// Brief: setup Arm Joint3-5 decelerate to stop
FUNCTION_BLOCK PUBLIC FB_SetupCtrlStop EXTENDS FB_SetupArmCtrlBase
VAR
	// stop motion is terminated after set time period
	m_maxStopPeriod :LREAL := 0.12;
	
	// deceleration period 
	m_decPeriod :LREAL := 0.1;

END_VAR

// override this function in each exact controller
METHOD PROTECTED calcCmdJntPos : BOOL
VAR_IN_OUT CONSTANT
	i_setupArm	:FB_SetupArm;
END_VAR


VAR 
	i :INT;
	nextCmdVel :LREAL;
END_VAR
IF m_isFinished THEN
	m_cmdJntVel := g_zeroVec5d;
	m_cmdJntPos := i_setupArm.curJntPos;
	RETURN;
END_IF

IF m_timePeriod > m_maxStopPeriod  THEN
	m_isFinished := TRUE;
	RETURN;
END_IF

FOR i := 3 TO 5 DO
	IF m_timePeriod > m_decPeriod THEN
		m_cmdJntVel[i] := 0;
	ELSE
		nextCmdVel := m_cmdJntVel[i] + m_cmdJntAcc[i]*g_setupArmCtrlCycleTime;
		m_cmdJntPos[i] := m_cmdJntPos[i] + (nextCmdVel + m_cmdJntVel[i])*g_setupArmCtrlCycleTime/2.0;
		m_cmdJntVel[i] := nextCmdVel;
	END_IF
END_FOR
END_METHOD

METHOD PUBLIC init : BOOL
VAR_IN_OUT CONSTANT
	i_setupArm	:FB_SetupArm;
END_VAR
VAR_IN_OUT 
	r_setupArmCtrlCmd :ST_SetupArmCtrlCmds;
END_VAR
VAR
	i:INT;
	maxJntTrq:LREAL;
END_VAR
// check if to hold the command joint position unchanged
m_holdLastCmds := checkToHoldLastCmds(i_setupArm);
SUPER^.Init(i_setupArm,r_setupArmCtrlCmd);

m_jntEnableFlag :=g_zeroVec5i;// setup arm joint is diabled by default

// determine joint deceleration
FOR i:=3 TO 5 DO 
		m_jntOPMode[i] := DriverOPMode_Pos;
		m_cmdJntVel[i] := i_setupArm.curJntVel[i];
		m_cmdJntAcc[i] := -i_setupArm.curJntVel[i]/m_decPeriod;
		m_jntEnableFlag[i] := BOOL_TO_INT(r_setupArmCtrlCmd.m_jntEnableFlag[i]=1 AND (r_setupArmCtrlCmd.m_jntOPMode[i] = DriverOPMode_Pos OR r_setupArmCtrlCmd.m_jntOPMode[i] = DriverOPMode_PosTrq));
END_FOR

IF m_jntEnableFlag[3] = 0 THEN
	m_jntOPMode[3]:= DriverOPMode_Trq;
END_IF
END_METHOD

END_FUNCTION_BLOCK

(* stored: Version 1.1.0.1, ProductVersion 3.1.4024.12
   POU FB_SetupCtrlStop: Id {2b39a0dc-24d1-457b-943f-73080894e676}, SpecialFunc None
   Method calcCmdJntPos: Id {7d3d4bc6-a9ba-43c5-8aaa-4916905417fa}
   Method init: Id {1aa46783-fabc-41be-a8ea-91f8151acc74} *)
